{attribute 'GeneratedUsingTerminal: EL3681-0000-0018'}
{attribute addProperty BoxType "EL3681-0000-0018"}
{attribute addProperty Id "StatusAT %I*Status_51F0A92410ValueAT %I*DINT4"}
{attribute addProperty CRC "2226298857"}
{attribute addProperty Size "14"}
TYPE SAI_Inputs_84B29FE9 :
STRUCT
	{attribute addProperty Name "Status"}
	Status AT %I* : Status_51F0A924;
	{attribute addProperty Name "Value"}
	Value AT %I* : DINT;
END_STRUCT
END_TYPE

(* stored: Version 1.2.0.0, ProductVersion 3.1.4024.9
   DUT SAI_Inputs_84B29FE9: Id {168ce242-606a-4b8e-a5c7-e395d5826956} *)
